# EPICS autosave request: asApp/Db/sample_settings.req
$(P)$(N).DRVH
$(P)$(N).DRVL
